{attribute 'linkalways'} 
{attribute 'no_explicit_call' := 'This FB is a CLASS and must be accessed using methods or properties'}
{attribute 'enable_dynamic_creation'}
FUNCTION_BLOCK _ETcVnContoursMatchComparisonMethod EXTENDS EnumDatatypeBase
VAR
	localData : ETcVnContoursMatchComparisonMethod;
	activeData : REFERENCE TO ETcVnContoursMatchComparisonMethod;
	enumBaseDatatype : _DINT(localData);
END_VAR

METHOD PRIVATE AddLocalEnumeration
VAR_INPUT
	Enumeration : T_MAXSTRING;
	Value : ETcVnContoursMatchComparisonMethod;
END_VAR
AddEnumeration(Enumeration, Value);
END_METHOD

PROPERTY PUBLIC Address : PVOID
GET
Address := ADR(activeData);
END_GET
END_PROPERTY

METHOD PUBLIC ClearReference
VAR_INPUT
END_VAR
activeData REF= localData;
SetBaseDatatypeReference();
END_METHOD

METHOD PUBLIC Clone : I_Datatype
VAR
    pClone : POINTER TO _ETcVnContoursMatchComparisonMethod;
END_VAR
pClone := __NEW(_ETcVnContoursMatchComparisonMethod(InitialValue := Value));
Clone := pClone^;
END_METHOD

METHOD FB_init : BOOL
VAR_INPUT
	bInitRetains : BOOL; // if TRUE, the retain variables are initialized (warm start / cold start)
	bInCopyCode : BOOL;  // if TRUE, the instance afterwards gets moved into the copy code (online change)
	InitialValue : ETcVnContoursMatchComparisonMethod;
END_VAR
localData := InitialValue;
AddBaseDatatype(enumBaseDatatype);
ClearReference();

AddLocalEnumeration('TCVN_CMCM_CONTOURS_MATCH_I1', ETcVnContoursMatchComparisonMethod.TCVN_CMCM_CONTOURS_MATCH_I1);
AddLocalEnumeration('TCVN_CMCM_CONTOURS_MATCH_I2', ETcVnContoursMatchComparisonMethod.TCVN_CMCM_CONTOURS_MATCH_I2);
AddLocalEnumeration('TCVN_CMCM_CONTOURS_MATCH_I3', ETcVnContoursMatchComparisonMethod.TCVN_CMCM_CONTOURS_MATCH_I3);
END_METHOD

PROPERTY PUBLIC Identifier : T_MAXSTRING
GET
Identifier := 'ETcVnContoursMatchComparisonMethod';
END_GET
END_PROPERTY

METHOD IsEnumeratorValueEqual : BOOL
VAR_INPUT
	Enumerator : I_KeyValueForwardEnumerator;
END_VAR
VAR
	storedValue : ETcVnContoursMatchComparisonMethod;
END_VAR
IF NOT Enumerator.TryGet(storedValue) THEN
	RETURN;
END_IF

IsEnumeratorValueEqual := storedValue = activeData;
END_METHOD

METHOD PUBLIC MakeReferenceTo
VAR_INPUT
	ReferenceTarget : REFERENCE TO ETcVnContoursMatchComparisonMethod;
END_VAR
activeData REF= ReferenceTarget;
SetBaseDatatypeReference();
END_METHOD

METHOD PROTECTED SetBaseDatatypeReference
VAR_INPUT
END_VAR
enumBaseDatatype.MakeReferenceTo(activeData);
END_METHOD

PROPERTY PUBLIC Size : UDINT
GET
Size := SIZEOF(activeData);
END_GET
END_PROPERTY

METHOD TryMakeReferenceTo : BOOL
VAR_INPUT
	Target : I_Datatype;
END_VAR
VAR
	targetAsEnum : I_EnumDatatype;
	pTargetData : POINTER TO ETcVnContoursMatchComparisonMethod;
END_VAR
IF NOT Target.TryResolveAsEnumDatatype(targetAsEnum) THEN
	RETURN;
END_IF

IF targetAsEnum.Identifier <> Identifier THEN
	RETURN;
END_IF

pTargetData := Target.Address;
activeData REF= pTargetData^;
SetBaseDatatypeReference();
TryMakeReferenceTo := TRUE;
END_METHOD

PROPERTY PUBLIC Value : ETcVnContoursMatchComparisonMethod
GET
Value := activeData;
END_GET
SET
activeData := Value;
END_SET
END_PROPERTY

END_FUNCTION_BLOCK

(* stored: Version 1.1.0.1
   POU _ETcVnContoursMatchComparisonMethod: Id {4228c25c-2e53-4ef8-a693-3c8142969087}, SpecialFunc None
   Folder Constructor: Id {62795e6e-7c69-43dd-a9fe-208c2452afba}
   Folder Private: Id {05bf6b58-59f4-480a-8ed9-71869a0d2628}
   Folder Protected: Id {aca55c9b-5c21-407d-ab85-5bdb33e27337}
   Method AddLocalEnumeration: Id {8bc3c848-250c-43b5-b0bb-fe8df877150a}
   Property Address: Id {60ee8a0c-4eb5-4d9d-b735-df29d8484b87}
   Get Get: Id {4323f330-161f-4cf2-8fce-196802b70790}
   Method ClearReference: Id {422af8c2-0b96-4531-9e18-cb3d8ba17538}
   Method Clone: Id {6f02f537-e6ae-4174-b7f8-9c41c6d457b6}
   Method FB_init: Id {41636535-a4d9-4be2-8649-7bd365b62713}
   Property Identifier: Id {e27b17d6-9b83-405f-a015-fa6825d6f855}
   Get Get: Id {24ff7a3e-210c-4f02-bfba-a722c4071f40}
   Method IsEnumeratorValueEqual: Id {cd1b4df4-2113-40cb-a4e6-631bbda26080}
   Method MakeReferenceTo: Id {1dffd1e3-11b5-47c4-8269-9f0398f25872}
   Method SetBaseDatatypeReference: Id {6949831a-c7bc-4bf8-b035-56113495158a}
   Property Size: Id {b39de8c7-286b-4339-b205-d989c10dc0d4}
   Get Get: Id {285ada65-2f67-4669-8a8d-1c718b8dc5b3}
   Method TryMakeReferenceTo: Id {557c67eb-9836-414f-a053-2b4158e043d0}
   Property Value: Id {d7657238-e63b-4dc0-89c0-2ccb821f3be8}
   Get Get: Id {96a4ee09-8428-434c-ae4e-b92579db610a}
   Set Set: Id {019f70f3-ce63-43fc-bf97-9bdef536ebed} *)
